(* LS Electric XG5000 project: 신호등_실습 *)
(* PLC LSPLC *)

PROGRAM NewProgram (* task: 스캔 프로그램 *)
VAR
    a : BOOL;
    q : BOOL;
    r : BOOL;
    set : BOOL;
    t1 : TON;
    t2 : TON;
    t3 : TP;
    t4 : TP;
    t5 : TON;
    t6 : TON;
    t7 : CTU_INT;
    t8 : CTD_INT;
    버튼 AT %MX0 : BOOL;
    차선_적색 AT %MX3 : BOOL;
    차선_청색 AT %MX1 : BOOL;
    차선_황색 AT %MX2 : BOOL;
    횡단보도_적색 AT %MX5 : BOOL;
    횡단보도_청색 AT %MX4 : BOOL;
END_VAR
VAR
    _e1 : R_TRIG;
    _p2 : BOOL;
    _e3 : R_TRIG;
END_VAR

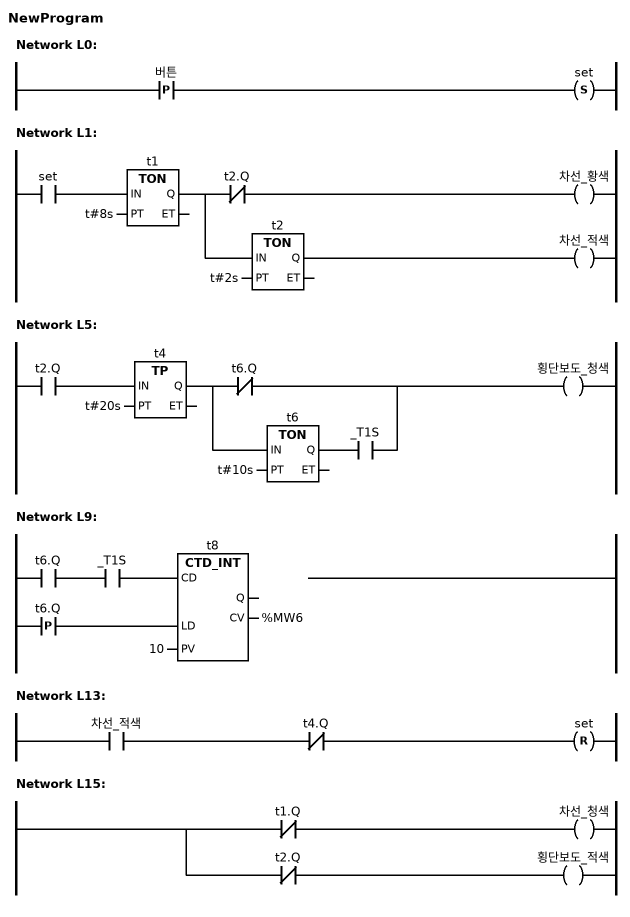
(* Rung L0 *)
_e1(CLK := 버튼);
IF _e1.Q THEN set := TRUE; END_IF;
(* Rung L1 *)
t1(IN := set, PT := t#8s);
차선_황색 := t1.Q AND NOT t2.Q;
t2(IN := t1.Q, PT := t#2s);
차선_적색 := t2.Q;
(* Rung L5 *)
t4(IN := t2.Q, PT := t#20s);
_p2 := t4.Q AND NOT t6.Q;
t6(IN := t4.Q, PT := t#10s);
횡단보도_청색 := _p2 OR (t6.Q AND _T1S);
(* Rung L9 *)
_e3(CLK := t6.Q);
t8(CD := t6.Q AND _T1S, LD := _e3.Q, PV := 10, CV => %MW6);
(* Rung L13 *)
IF 차선_적색 AND NOT t4.Q THEN set := FALSE; END_IF;
(* Rung L15 *)
차선_청색 := NOT t1.Q;
횡단보도_적색 := NOT t2.Q;
END_PROGRAM